
(* ===== HMI "HMI_RT_1" =====

HMI tags "email"
   "_EMAIL_" : 22c219e6-cff3-42c5-8b54-d29671cf4baa, internal
   "_SMTP_" : 9be4dde3-9bf9-494b-8378-d23bba93c127, internal
*)